SEGMENT_TYPE PROFInet (* PROFInet Segment *)
  (* Standard: 61499 ITA; Description: PROFInet ... *)
  (* Version 0.0, 2008-07-10, 4DIAC-IDE, 4DIAC-Consortium *)
  VAR_INPUT
    Param : WSTRING; (* Param *)
  END_VAR
END_SEGMENT_TYPE
